# B&R Automation Studio project ULATolo3
Automation Studio 4.7.5.60 SP; technology packages: mapp 5.11.2, mappMotion 5.11.2

## Configuration Config1

CPU X20CP1382, AutomationRuntime B4.73, Build 4.1.2, Safety 0.0, Vc V4.72.0

### Task classes (Cpu.sw)
```
Cyclic#1 (cycle 1200 us, tolerance 0 us):
  Program <- Program.prg
DataObjects: ALHistory
VcDataObjects: Visu <- Visu.dob
Binaries: vccdt, vccbmp, Visu03, vcfile, arial, vccddbox, vcrt, vccstr, vcbclass, vccbtn, vcgclass, vcdsint, vcnet, vccline, vcmgr, vcshared, vcclbox, vccscale, arialbd, vccnum, vcpdvnc, FWRules, vccalarm, vccshape, vcctext, Visu01, vcpdsw, vcfntttf, vccovl, vcalarm, vcpkat, Visu02, udbdef, vccpopup, arsvcreg, vcdsloc, vcchspot, vctcal, TCData, vcpfx20, Config, arconfig, Config_1, asfw, iomap, Role, ashwd, ashwac, sysconf, User, vcpfar00
Libraries: brsystem, sys_lib, runtime, MpAxis, MpCom, MpBase, MpAlarmX, astime, AsBrStr, McBase, McAxis, McAcpAx, asieccon, powerlnk, vcresman, ashw, MpData, DataObj, FileIO
```

### Hardware
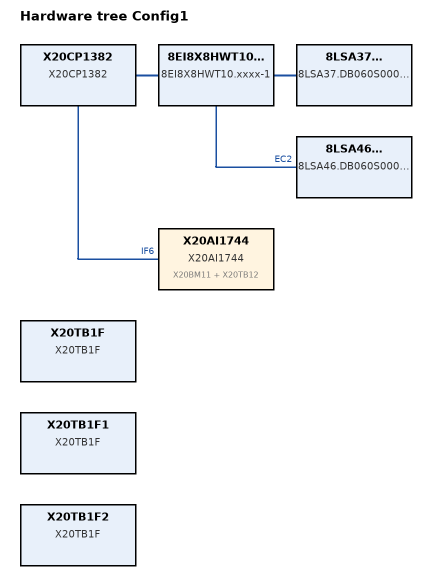
```
8EI8X8HWT10.xxxx-1 : 8EI8X8HWT10.xxxx-1 v2.3.0.3  [PLK2 -> X20CP1382.IF3 [Cable Type=PowerlinkCable, Length=10, Version=1.0.0.2]; EC1 -> 8LSA37.DB060S000-3a.EC; EC2 -> 8LSA46.DB060S000-3.EC; MT2 -> 8LSA46.DB060S000-3.MT]
  MotionTP = Acp10Arnc0
  EnableDNA = on
  EPL_DNA_Head = 0
  EPL_DNA_HubPort = 1
  DriveConfiguration/Module:
    McAcoposTypeID = AcoposP3TConfig
    ActivateACOPOSSimulationOnPLC = 0
  DriveConfiguration/Encoder/EncoderX41:
    InterfaceType = EnDat
  DriveConfiguration/Encoder/EncoderX42:
    InterfaceType = EnDat
  DriveConfiguration/Channel[1]:
    License = 1
  DriveConfiguration/Channel[1]/RealAxis:
    AxisReference = gAxisBasicAxial
  DriveConfiguration/Channel[1]/RealAxis/MechanicalElements/Gearbox:
    InputIsReadOnly = 0
    Input = 40
    OutputIsReadOnly = 0
    Output = 1
  DriveConfiguration/Channel[1]/RealAxis/MechanicalElements/RotaryToLinearTransformation:
    ReferenceDistanceIsReadOnly = 0
    ReferenceDistance = 12.7
  DriveConfiguration/Channel[1]/RealAxis/Controller:
    ModeIsReadOnly = 0
    Mode = PositionController
  DriveConfiguration/Channel[1]/RealAxis/Controller/Mode/Position:
    ProportionalGain = 430
    IntegrationTime = 0.0
    PredictionTime = 0.0004
    TotalDelayTime = 0.0004
  DriveConfiguration/Channel[1]/RealAxis/Controller/Mode/Speed:
    ProportionalGainIsReadOnly = 0
    ProportionalGain = 2.9
    IntegrationTimeIsReadOnly = 0
    IntegrationTime = 0.0
    FilterTimeIsReadOnly = 0
    FilterTime = 0.0
  DriveConfiguration/Channel[1]/RealAxis/Controller/Mode/LoopFilters:
    LoopFilter1 = NotUsed
    LoopFilter2 = NotUsed
    LoopFilter3 = NotUsed
  DriveConfiguration/Channel[1]/RealAxis/Homing:
    Mode = Absolute
  DriveConfiguration/Channel[1]/RealAxis/Homing/Mode:
    Position = 1238.54
  DriveConfiguration/Channel[1]/RealAxis/Homing:
    RestorePositionVariable = 
  DriveConfiguration/Channel[1]/RealAxis/StopReaction:
    Quickstop = DecelerationLimit
    DriveError = DecelerationLimit
  DriveConfiguration/Channel[1]/RealAxis/MovementErrorLimits:
    PositionError = 1.0
    VelocityErrorMonitoring = Automatic1
  DriveConfiguration/Channel[1]/RealAxis:
    JerkFilter = NotUsed
  DriveConfiguration/Channel[1]/RealAxis/DigitalInputs/HomingSwitch:
    Source = NotUsed
    Level = High
  DriveConfiguration/Channel[1]/RealAxis/DigitalInputs/PositiveLimitSwitch:
    Source = NotUsed
    Level = High
  DriveConfiguration/Channel[1]/RealAxis/DigitalInputs/NegativeLimitSwitch:
    Source = NotUsed
    Level = High
  DriveConfiguration/Channel[1]/RealAxis/DigitalInputs/Trigger1:
    Source = X8Trigger1
    Level = High
  DriveConfiguration/Channel[1]/RealAxis/DigitalInputs/Trigger2:
    Source = X8Trigger2
    Level = High
  DriveConfiguration/Channel[1]/RealAxis/DigitalInputs/Quickstop:
    Input = Trigger2
  DriveConfiguration/Channel[1]/RealAxis/Simulation:
    SimulationModeOnPLC = SetValueGeneration
    SimulationModeOnACOPOS = NotUsed
  DriveConfiguration/Channel[2]:
    License = 1
  DriveConfiguration/Channel[2]/RealAxis:
    AxisReference = gAxisBasicSideLoad
  DriveConfiguration/Channel[2]/RealAxis/MechanicalElements/Gearbox:
    InputIsReadOnly = 0
    Input = 1
    OutputIsReadOnly = 0
    Output = 1
  DriveConfiguration/Channel[2]/RealAxis/MechanicalElements/RotaryToLinearTransformation:
    ReferenceDistanceIsReadOnly = 0
    ReferenceDistance = 1
  DriveConfiguration/Channel[2]/RealAxis/Controller:
    ModeIsReadOnly = 0
    Mode = PositionController
  DriveConfiguration/Channel[2]/RealAxis/Controller/Mode/Position:
    ProportionalGain = 50.0
    IntegrationTime = 0.0
    PredictionTime = 0.0004
    TotalDelayTime = 0.0004
  DriveConfiguration/Channel[2]/RealAxis/Controller/Mode/Speed:
    ProportionalGainIsReadOnly = 0
    ProportionalGain = 2.0
    IntegrationTimeIsReadOnly = 0
    IntegrationTime = 0.0
    FilterTimeIsReadOnly = 0
    FilterTime = 0.0
  DriveConfiguration/Channel[2]/RealAxis/Controller/Mode/LoopFilters:
    LoopFilter1 = NotUsed
    LoopFilter2 = NotUsed
    LoopFilter3 = NotUsed
  DriveConfiguration/Channel[2]/RealAxis/Homing:
    Mode = Absolute
  DriveConfiguration/Channel[2]/RealAxis/Homing/Mode:
    Position = 12888.441
  DriveConfiguration/Channel[2]/RealAxis/Homing:
    RestorePositionVariable = 
  DriveConfiguration/Channel[2]/RealAxis/StopReaction:
    Quickstop = DecelerationLimit
    DriveError = DecelerationLimit
  DriveConfiguration/Channel[2]/RealAxis/MovementErrorLimits:
    PositionError = 1.0
    VelocityErrorMonitoring = Automatic1
  DriveConfiguration/Channel[2]/RealAxis:
    JerkFilter = NotUsed
  DriveConfiguration/Channel[2]/RealAxis/DigitalInputs/HomingSwitch:
    Source = NotUsed
    Level = High
  DriveConfiguration/Channel[2]/RealAxis/DigitalInputs/PositiveLimitSwitch:
    Source = NotUsed
    Level = High
  DriveConfiguration/Channel[2]/RealAxis/DigitalInputs/NegativeLimitSwitch:
    Source = NotUsed
    Level = High
  DriveConfiguration/Channel[2]/RealAxis/DigitalInputs/Trigger1:
    Source = X8Trigger1
    Level = High
  DriveConfiguration/Channel[2]/RealAxis/DigitalInputs/Trigger2:
    Source = X8Trigger2
    Level = High
  DriveConfiguration/Channel[2]/RealAxis/DigitalInputs/Quickstop:
    Input = Trigger2
  DriveConfiguration/Channel[2]/RealAxis/Simulation:
    SimulationModeOnPLC = SetValueGeneration
    SimulationModeOnACOPOS = NotUsed
  DriveConfiguration/Channel[3]:
    License = 1
  DriveConfiguration/Channel[3]/RealAxis:
    AxisReference = 
  DriveConfiguration/Channel[3]/RealAxis/MechanicalElements/Gearbox:
    InputIsReadOnly = 0
    Input = 1
    OutputIsReadOnly = 0
    Output = 1
  DriveConfiguration/Channel[3]/RealAxis/MechanicalElements/RotaryToLinearTransformation:
    ReferenceDistanceIsReadOnly = 0
    ReferenceDistance = 1
  DriveConfiguration/Channel[3]/RealAxis/Controller:
    ModeIsReadOnly = 0
    Mode = PositionController
  DriveConfiguration/Channel[3]/RealAxis/Controller/Mode/Position:
    ProportionalGain = 50.0
    IntegrationTime = 0.0
    PredictionTime = 0.0004
    TotalDelayTime = 0.0004
  DriveConfiguration/Channel[3]/RealAxis/Controller/Mode/Speed:
    ProportionalGainIsReadOnly = 0
    ProportionalGain = 2.0
    IntegrationTimeIsReadOnly = 0
    IntegrationTime = 0.0
    FilterTimeIsReadOnly = 0
    FilterTime = 0.0
  DriveConfiguration/Channel[3]/RealAxis/Controller/Mode/LoopFilters:
    LoopFilter1 = NotUsed
    LoopFilter2 = NotUsed
    LoopFilter3 = NotUsed
  DriveConfiguration/Channel[3]/RealAxis/Homing:
    Mode = Direct
  DriveConfiguration/Channel[3]/RealAxis/Homing/Mode:
    Position = 0.0
    ReferencePulse = NotUsed
  DriveConfiguration/Channel[3]/RealAxis/Homing:
    RestorePositionVariable = 
  DriveConfiguration/Channel[3]/RealAxis/StopReaction:
    Quickstop = DecelerationLimit
    DriveError = DecelerationLimit
  DriveConfiguration/Channel[3]/RealAxis/MovementErrorLimits:
    PositionError = 1.0
    VelocityErrorMonitoring = Automatic1
  DriveConfiguration/Channel[3]/RealAxis:
    JerkFilter = NotUsed
  DriveConfiguration/Channel[3]/RealAxis/DigitalInputs/HomingSwitch:
    Source = NotUsed
    Level = High
  DriveConfiguration/Channel[3]/RealAxis/DigitalInputs/PositiveLimitSwitch:
    Source = NotUsed
    Level = High
  DriveConfiguration/Channel[3]/RealAxis/DigitalInputs/NegativeLimitSwitch:
    Source = NotUsed
    Level = High
  DriveConfiguration/Channel[3]/RealAxis/DigitalInputs/Trigger1:
    Source = X8Trigger1
    Level = High
  DriveConfiguration/Channel[3]/RealAxis/DigitalInputs/Trigger2:
    Source = X8Trigger2
    Level = High
  DriveConfiguration/Channel[3]/RealAxis/DigitalInputs/Quickstop:
    Input = Trigger2
  DriveConfiguration/Channel[3]/RealAxis/Simulation:
    SimulationModeOnPLC = SetValueGeneration
    SimulationModeOnACOPOS = NotUsed
8LSA37.DB060S000-3a : 8LSA37.DB060S000-3 v1.0.5.34  [EC -> 8EI8X8HWT10.xxxx-1.EC1; MT -> 8EI8X8HWT10.xxxx-1.MT1]
8LSA46.DB060S000-3 : 8LSA46.DB060S000-3 v2.2.0.0  [EC -> 8EI8X8HWT10.xxxx-1.EC2; MT -> 8EI8X8HWT10.xxxx-1.MT2]
  M1/MotorParameters:
    MOTOR_AMB_TEMP_RATED = 40
  M1/MotorParameters/TemperatureSensor:
    MOTOR_TEMPSENS_LIM = 130
X20AI1744 : X20AI1744 v1.8.4.0  [SS1 -> X20TB12.SS; SL -> X20BM11.SL1]
  Supervision = off
X20BM11 : X20BM11 v1.0.0.1  [X2X1 -> X20CP1382.IF6]
X20CP1382 : X20CP1382 v1.8.0.0  [X1 -> X1.SL; X2 -> X2.SL; X3 -> X3.SL]
  Module X1 (Type=X1, Virtual=true, Version=1.8.0.0)
    Connection (Connector=SS1, TargetModule=X20TB1F, TargetConnector=SS)
    Connection (Connector=SL, TargetModule=X20CP1382, TargetConnector=X1)
  Module X2 (Type=X2, Virtual=true, Version=1.8.0.0)
    Connection (Connector=SS1, TargetModule=X20TB1F1, TargetConnector=SS)
    Connection (Connector=SL, TargetModule=X20CP1382, TargetConnector=X2)
  Module X3 (Type=X3, Virtual=true, Version=1.8.0.0)
    Connection (Connector=SS1, TargetModule=X20TB1F2, TargetConnector=SS)
    Connection (Connector=SL, TargetModule=X20CP1382, TargetConnector=X3)
  Connector IF2:
    ActivateDevice = 1
    Mode = Manual
    InternetAddress = 192.168.1.5
    SubnetMask = 255.255.255.0
    Vnc1
    VncVcObjectName1 = Visu
    VncKeyMappingFile1 = VC\PS2-Keyboard.dis
  Connector IF3:
    CycleTime = 1200
  ConfigurationID = ULATolo3_Config1
  Simulation = 1
  VolatileGlobalPvSize = 6553500
  TimerDeviceType = EPLX2X
  TimerDevice = X20CP1382.IF3
  TaskClassIdleTime = 9600
  Cyclic1Duration = 1200
  Cyclic1Tolerance = 0
  Cyclic1Stack = 65535
  Cyclic2Duration = 20400
  Cyclic2Tolerance = 20400
  Cyclic3Duration = 50400
  Cyclic3Tolerance = 50400
  Cyclic4Duration = 99600
  Cyclic4Tolerance = 99600
  Cyclic5Duration = 200400
  Cyclic5Tolerance = 200400
  Cyclic6Duration = 500400
  Cyclic6Tolerance = 500400
  Cyclic7Duration = 999600
  Cyclic7Tolerance = 999600
  Cyclic8Duration = 9600
  FileDevice1
  FileDeviceName1 = Temp
  FileDevicePath1 = C:\Temp
  FileDevice2
  FileDeviceName2 = PLC
  FileDevicePath2 = F:\
X20TB12 : X20TB12 v1.0.0.0
X20TB1F : X20TB1F v1.0.0.0
X20TB1F1 : X20TB1F v1.0.0.0
X20TB1F2 : X20TB1F v1.0.0.0
```

### IoMap.iom - X20CP1382/IoMap.iom
```iecst
VAR_CONFIG
	::gMain.Input.Physical.StrainGauge AT %ID."X20AI1744".AnalogInput01;
	::gMain.Machine.Motion.PosLimit AT %IX."X1".DigitalInput01;
	::gMain.Machine.Motion.NegLimit AT %IX."X1".DigitalInput02;
END_VAR
```

### Acp10cfg.ncc - X20CP1382/Motion/Acp10cfg.ncc
```
NcConfiguration (Version=5.08.2, NcSwId=Acp10)
  ACP10CF1_typ:
    cnt_nettrc_rec_drive = 1500
    bufsize_trace_upload = 1200
    tc_nc_man_task = Cyclic #1
    glob_pv_as_ncobject = Yes
    ncsys_dl_broadcast = Yes
    ncsys_dl_acp_reset = Yes
    safemc_log_err_to_ax = Yes
    network_init:
      ncsw_init_execute = Yes
      automatic_execute = No
      node_nr_warning = Yes
      net_err_before_ncact = Yes
    nettrc:
      enter_parsecrec = Yes
      enter_ncaction = Yes
      save_ring_startidx = Yes
    cam_prof_download:
      cam_dat_dl_parallel = No
      tc_cam_dl_parallel = Task class for NC Manager task
    plk_if[0]:
      if_name = IF3
      tc_CycDat_PLCopen = Task class for NC Manager task
      mc_broadcast_extdat = No
```

### Acp10map.ncm - X20CP1382/Motion/Acp10map.ncm
```
NcMapping (NcSwId=Acp10, DisabledNodesAreHidden=False)
  NcObject gAxisSideLoad (ModuleId=8EI8X8HWT10.xxxx-1, Type=ncAXIS, Channel=2, AcoposSimulation=Off, InitParameter=gAxis01i, AcoposParameter=gAxis01a, Disabled=FALSE, ModuleDisabled=FALSE)
  NcObject gAxisAxial (ModuleId=8EI8X8HWT10.xxxx-1, Type=ncAXIS, Channel=1, AcoposSimulation=Off, InitParameter=gAxis01i, AcoposParameter=gAxis01a, Disabled=FALSE, ModuleDisabled=FALSE)
  NcObject 8EI4X5HWD10.xxxx-1_ncAXIS3 (ModuleId=8EI8X8HWT10.xxxx-1, Type=ncAXIS, Channel=3, AcoposSimulation=off, Disabled=true, ModuleDisabled=FALSE)
  NcObject 8EI4X5HWD10.xxxx-1_ncV_AXIS2 (ModuleId=8EI8X8HWT10.xxxx-1, Type=ncV_AXIS, Channel=2, Disabled=TRUE, ModuleDisabled=FALSE)
  NcObject 8EI4X5HWD10.xxxx-1_ncV_AXIS1 (ModuleId=8EI8X8HWT10.xxxx-1, Type=ncV_AXIS, Channel=1, Disabled=TRUE, ModuleDisabled=FALSE)
  NcObject 8EI4X5HWD10.xxxx-1_ncV_AXIS3 (ModuleId=8EI8X8HWT10.xxxx-1, Type=ncV_AXIS, Channel=3, AcoposSimulation=off, Disabled=true, ModuleDisabled=FALSE)
```

### Config.mpaxisbasic - X20CP1382/Motion/Config.mpaxisbasic
```
Element gAxisBasicAxial (Type=mpaxisbasic)
  AxisConfiguration = AxisWithConfiguration
    Axis:
      BaseType = 4
      MeasurementUnit = 1
      PeriodSettings:
        Period = 360
      MovementLimits:
        VelocityPositive = 10000.0
        VelocityNegative = 10000.0
        Acceleration = 50000.0
        Deceleration = 50000
        JerkTime = 0.01
        PositionErrorStopLimit = 1000
    Drive:
      Transformation:
        ReferenceDistance = 12.7
      Controller:
        LoopFilters:
          [0]
          [1]
          [2]
  Alarms = MpAlarmX
Element gAxisBasicSideLoad (Type=mpaxisbasic)
  Alarms = MpAlarmX
```

### Axial.axis - X20CP1382/mappMotion/Axial.axis
```
Element gAxisBasicAxial (Type=axis)
  BaseTypeIsReadOnly = 0
  BaseType = LinearBounded
    MeasurementUnit = 5066068
    MeasurementResolutionIsReadOnly = 0
    MeasurementResolution = 0.01
    CountDirectionIsReadOnly = 0
    CountDirection = Standard
  MovementLimitsIsReadOnly = 0
  MovementLimits = Internal
    Position:
      LowerLimitMin = -1.79769313486231E308
      UpperLimitMax = 1.79769313486231E308
      LowerLimit = 388.62
      UpperLimit = 608.6348
    VelocityIsReadOnly = 0
    Velocity:
      VelocityMax = 3.4E38
      Velocity = 50
    AccelerationIsReadOnly = 0
    Acceleration:
      AccelerationMax = 3.4E38
      Acceleration = 75
    DecelerationIsReadOnly = 0
    Deceleration:
      DecelerationMax = 3.4E38
      Deceleration = 75
  Alarms = MpAlarmX
```

### Side.axis - X20CP1382/mappMotion/Side.axis
```
Element gAxisBasicSideLoad (Type=axis)
  BaseTypeIsReadOnly = 0
  BaseType = LinearBounded
    MeasurementUnit = 5066068
    MeasurementResolutionIsReadOnly = 0
    MeasurementResolution = 0.01
    CountDirectionIsReadOnly = 0
    CountDirection = Standard
  MovementLimitsIsReadOnly = 0
  MovementLimits = Internal
    Position:
      LowerLimitMin = -1.79769313486231E308
      UpperLimitMax = 1.79769313486231E308
      LowerLimit = -1000.0
      UpperLimit = 1000.0
    VelocityIsReadOnly = 0
    Velocity:
      VelocityMax = 3.4E38
      Velocity = 25
    AccelerationIsReadOnly = 0
    Acceleration:
      AccelerationMax = 3.4E38
      Acceleration = 75
    DecelerationIsReadOnly = 0
    Deceleration:
      DecelerationMax = 3.4E38
      Deceleration = 75
  Alarms = MpAlarmX
```

### Config.mpdatarecorder - X20CP1382/mappServices/Config.mpdatarecorder
```
Element gDataRecorder (Type=mpdatarecorder)
  Alarms = MpAlarmX
```

### Config_1.mpalarmxcore - X20CP1382/mappServices/Config_1.mpalarmxcore
```
Element gAlarmXCore (Type=mpalarmxcore)
```

## Logical view

Binary libraries used (declarations not repeated): operator, runtime, astime, AsIecCon, brsystem, sys_lib, AsBrStr, McBase 5.11.2, McAxis 5.11.2, MpBase 5.11.0, MpAlarmX 5.11.2, MpCom 5.11.2, MpAxis 5.11.2, McAcpAx 5.11.2, MpData 5.11.2, DataObj, FileIO, Acp10_MC 5.10.1, Acp10man 5.10.1, Acp10par 5.10.1, NcGlobal 5.10.1

### Global.typ - Global data types
```iecst
TYPE
	Alarm_Type : 	STRUCT
		MpAlarmXListUI_FB : MpAlarmXListUI;
		MpAlarmXAcknowledgeAll_FB : MpAlarmXAcknowledgeAll;
		MpAlarmXListUISetupType : MpAlarmXListUISetupType;
		MpAlarmXListUIConnectType : MpAlarmXListUIConnectType;
		AlarmPopupControl : USINT;
		MpAlarmXCore_FB : MpAlarmXCore;
	END_STRUCT;
	InputPhysical_Type : 	STRUCT
		LoadtoTorqueScaleFactor : REAL;
		StrainGauge : DINT;
	END_STRUCT;
	Output_Type : 	STRUCT
		Physical : OutputPhysical_Type;
		Vis : OutputVis_Type;
	END_STRUCT;
	OutputVis_Type : 	STRUCT
		DisplayedForceFeedback : REAL;
		StatusLED : USINT;
		LoadCellScaleFactor : REAL;
		CalculatedForce : REAL;
	END_STRUCT;
	OutputPhysical_Type : 	STRUCT
		New_Member : USINT;
	END_STRUCT;
	InputVis_Type : 	STRUCT
		NumberofCycles : USINT;
		ManualCommandedAxialPosition : REAL;
		ManualReturnButton : BOOL;
		ManualCommandedSideLoad : REAL;
		AxisSelector : USINT;
		JogNeg : BOOL;
		JogPos : BOOL;
		ManualMoveButton : BOOL;
		StartProgramButton : BOOL;
		NominalPosition : REAL;
		AutoCommandedAxialPosition : REAL;
		PowerOnButtonVisibility : USINT;
		JogButtonVisibility : USINT;
		StopButtonVisibility : USINT;
		StartButtonVisability : USINT;
		EStopPopup : USINT;
		EStop : BOOL;
		PowerOnAll : BOOL;
		OscillationDistance : REAL;
		ManualStopButtonVis : UINT;
		ConfirmPopup : USINT;
		ManualGoButtonVis : UINT;
	END_STRUCT;
	Input_Type : 	STRUCT
		Physical : InputPhysical_Type;
		Vis : InputVis_Type;
	END_STRUCT;
	Motion_Type : 	STRUCT
		MpAxisBasicPar : ARRAY[Axial..SideLoad]OF MpAxisBasicParType;
		Mc_StopFB : ARRAY[Axial..SideLoad]OF MC_Stop;
		MpAxisBasic_FB : ARRAY[Axial..SideLoad]OF MpAxisBasic;
		Error : BOOL;
		HomeAll : BOOL;
		IsHomedAll : BOOL;
		AllAxisReady : BOOL;
		ErrorResetAll : BOOL;
		SideLoad : SideLoad_Type;
		AxialMove : AxialMove_Type;
		IsPoweredAll : BOOL;
		AtNominalFlag : BOOL;
	END_STRUCT;
	Machine_Type : 	STRUCT
		State : StateEnum;
		Alarm : Alarm_Type;
		Motion : Motion_Type;
	END_STRUCT;
	Main_Type : 	STRUCT
		Output : Output_Type;
		Input : Input_Type;
		Machine : Machine_Type;
		Services : Services_Type;
	END_STRUCT;
	SideLoad_Type : 	STRUCT
		ScalingFactor : REAL;
		EnableCyclicTorque : BOOL;
		TorqueScaled : REAL;
		MC_TorqueControl_FB : MC_TorqueControl;
		MC_MoveAdditive_SideLoad : MC_MoveAdditive;
	END_STRUCT;
	AxialMove_Type : 	STRUCT
		Amax : REAL;
		TotalDistance : REAL;
		Vmax : REAL;
		TotalTime : REAL;
		CyclicCommandedPosition : REAL;
		CycleAmplitude : REAL;
		FirstMovementFlag : BOOL;
		ChangeDirectionFlag : BOOL;
		CycleCount : UDINT;
		PositionOffset : REAL;
		MC_MoveAdditive_Axial : MC_MoveAdditive;
	END_STRUCT;
	AxisEnum :
		(
		SideLoad := 1,
		Axial := 0
		);
	StateEnum :
		(
		Running := 6,
		Idle := 5,
		WaitingForPowerOn := 4,
		Homing := 3,
		AxisReady := 2,
		Init := 1,
		Error := 0
		);
	Services_Type : 	STRUCT
		MpDataRegPar : MpDataRegPar;
		MpDataRecorder_FB : MpDataRecorder;
	END_STRUCT;
END_TYPE
```

### Global.var - Global variables
```iecst
VAR
	gMain : Main_Type;
	i0 : USINT;
END_VAR
```

### Package Logical/Libraries - Global libraries

- Visualisation Logical/Visu (not shown)

### Program Logical/Program (IEC)

#### Variables.var
```iecst
VAR CONSTANT
	MAX_TORQUE : REAL := 169.477;
END_VAR
```

#### Main.st
```iecst
PROGRAM _INIT

//
//		gMain.Machine.Motion.AxialMove.CycleAmplitude:=12.7;
//		gMain.Machine.Motion.AxialMove.TotalTime:=0.0825;
//		gMain.Machine.Motion.AxialMove.TotalDistance:=gMain.Machine.Motion.AxialMove.CycleAmplitude*2;
//		gMain.Machine.Motion.AxialMove.PositionOffset:=18.2*25.4;
//
//	gMain.Machine.Motion.Mc_StopFB[Axial](Axis := ADR(gAxisAxial), Deceleration := 50000);
//	gMain.Machine.Motion.Mc_StopFB[SideLoad](Axis := ADR(gAxisSideLoad), Deceleration := 50000);
//
//		// Velocity AND Acceleration Calculations FOR Axial MOVE
//		IF gMain.Machine.Motion.AxialMove.TotalTime<>0.0 THEN
//			gMain.Machine.Motion.AxialMove.Vmax:=ABS(gMain.Machine.Motion.AxialMove.TotalDistance/(0.5*(gMain.Machine.Motion.AxialMove.TotalTime)));
//			gMain.Machine.Motion.AxialMove.Amax:=ABS(gMain.Machine.Motion.AxialMove.Vmax/(0.5*gMain.Machine.Motion.AxialMove.TotalTime));
//		END_IF;
//
//	gMain.Machine.Motion.MpAxisBasicPar[Axial].Acceleration:=gMain.Machine.Motion.AxialMove.Amax;
//	gMain.Machine.Motion.MpAxisBasicPar[Axial].Deceleration:=gMain.Machine.Motion.AxialMove.Amax;
//	gMain.Machine.Motion.MpAxisBasicPar[Axial].Velocity:=gMain.Machine.Motion.AxialMove.Vmax;
//
//
//
//	gMain.Machine.Motion.MpAxisBasicPar[Axial].Home.Mode:=mpAXIS_HOME_MODE_ABSOLUTE;
//	gMain.Machine.Motion.MpAxisBasicPar[Axial].Home.Position:=1238.54;						//0 position is -610.77
//
//	gMain.Machine.Motion.MpAxisBasicPar[SideLoad].Home.Mode:=mpAXIS_HOME_MODE_ABSOLUTE;
//	gMain.Machine.Motion.MpAxisBasicPar[SideLoad].Home.Position:=12888.441;

	gMain.Machine.Motion.MpAxisBasic_FB[Axial].MpLink := ADR(gAxisBasicAxial);
	gMain.Machine.Motion.MpAxisBasic_FB[Axial].Enable := TRUE;
	gMain.Machine.Motion.MpAxisBasic_FB[Axial].Parameters := ADR(gMain.Machine.Motion.MpAxisBasicPar[Axial]);
	//gMain.Machine.Motion.MpAxisBasic_FB[Axial].Axis := ADR(gAxisAxial);

	gMain.Machine.Motion.MpAxisBasic_FB[SideLoad].MpLink :=ADR(gAxisBasicSideLoad);
	gMain.Machine.Motion.MpAxisBasic_FB[SideLoad].Enable := TRUE;
	gMain.Machine.Motion.MpAxisBasic_FB[SideLoad].Parameters := ADR(gMain.Machine.Motion.MpAxisBasicPar[SideLoad]);
	//gMain.Machine.Motion.MpAxisBasic_FB[SideLoad].Axis := ADR(gAxisSideLoad);

	gMain.Machine.Motion.SideLoad.MC_TorqueControl_FB.Axis := ADR(gAxisBasicSideLoad);
	gMain.Machine.Motion.SideLoad.MC_TorqueControl_FB.TorqueRamp := 0.3;
	gMain.Machine.Motion.SideLoad.MC_TorqueControl_FB.Velocity := 10;
	gMain.Machine.Motion.SideLoad.MC_TorqueControl_FB.Acceleration := 10;

	gMain.Machine.Alarm.MpAlarmXCore_FB(MpLink :=ADR(gAlarmXCore),Enable := TRUE);
	gMain.Machine.Alarm.MpAlarmXListUI_FB(MpLink := ADR(gAlarmXCore), Enable := TRUE, UISetup := gMain.Machine.Alarm.MpAlarmXListUISetupType, UIConnect := ADR(gMain.Machine.Alarm.MpAlarmXListUIConnectType));

//	gMain.Machine.Motion.MpAxisBasicPar[SideLoad].CyclicRead.TorqueMode:=mpAXIS_READ_CYCLIC;

	gMain.Output.Vis.LoadCellScaleFactor:= (100.0/-307482);
	gMain.Machine.Motion.SideLoad.ScalingFactor := 0.0034;

	gMain.Machine.Motion.MpAxisBasicPar[Axial].Jog.Velocity:=25.4;

	//Data Logging
	gMain.Services.MpDataRecorder_FB.DeviceName := ADR('Temp');
	gMain.Services.MpDataRecorder_FB.RecordMode := mpDATA_RECORD_MODE_VALUE;
	gMain.Services.MpDataRecorder_FB.MpLink := ADR(gDataRecorder);
	gMain.Services.MpDataRecorder_FB.Enable :=  TRUE;

	gMain.Services.MpDataRegPar.MpLink := ADR(gDataRecorder);
	gMain.Services.MpDataRegPar.Enable := TRUE;
	gMain.Services.MpDataRegPar.PVName := ADR('gMain.Input.Vis.StartProgramButton');

	//Popup Vis
	gMain.Input.Vis.ConfirmPopup := TRUE;
END_PROGRAM

PROGRAM _CYCLIC
	gMain.Machine.Motion.AllAxisReady :=TRUE;
	gMain.Machine.Motion.IsHomedAll := TRUE;
	gMain.Machine.Motion.IsPoweredAll := TRUE;
	gMain.Machine.Motion.Error := FALSE;
	//gMain.Machine.Motion.AxialMove.MC_MoveAdditive_Axial.Execute:=FALSE;

	//Check State Loop
	FOR i0:=DINT_TO_USINT(Axial) TO DINT_TO_USINT(SideLoad) DO
		IF NOT gMain.Machine.Motion.MpAxisBasic_FB[i0].Info.ReadyToPowerOn AND NOT gMain.Machine.Motion.MpAxisBasic_FB[i0].Info.ReadyToPowerOn THEN //If not axis initilaized and not ready to power on
			gMain.Machine.Motion.AllAxisReady := FALSE;  																						   //Then set DrivesReady to FALSE
		END_IF;
		IF gMain.Machine.Motion.MpAxisBasic_FB[i0].IsHomed = FALSE THEN																				//If single axis is not homed
			gMain.Machine.Motion.IsHomedAll := FALSE;																								//Then IsHomedAll is FALSE
		END_IF;
		IF gMain.Machine.Motion.MpAxisBasic_FB[i0].PowerOn = FALSE THEN																				//If drive PowerOn is FALSE for single axis
			gMain.Machine.Motion.IsPoweredAll := FALSE;																								//Then IsPoweredAll is FALSE
		END_IF;
		IF gMain.Machine.Motion.MpAxisBasic_FB[i0].Error THEN
			gMain.Machine.Motion.Error:=TRUE;
		END_IF;
	END_FOR;

	//Machine State Case Statement
	CASE gMain.Machine.State OF
		Error:
			IF gMain.Machine.Motion.Error THEN
			ELSE
				gMain.Machine.State:=Init;
			END_IF;
			gMain.Input.Vis.PowerOnAll:=FALSE;
			gMain.Output.Vis.StatusLED:=0;
			gMain.Services.MpDataRecorder_FB.Record := FALSE;
		Init:
			IF gMain.Machine.Motion.Error THEN
				gMain.Machine.State:=Error;
			ELSIF gMain.Machine.Motion.AllAxisReady THEN
				gMain.Machine.Motion.HomeAll:=TRUE;
				gMain.Machine.State:=Homing;
			END_IF;
		Homing:
			IF gMain.Machine.Motion.Error THEN
				gMain.Machine.State:=Error;
			ELSIF gMain.Machine.Motion.IsHomedAll THEN
				gMain.Machine.Motion.HomeAll:=FALSE;
				gMain.Machine.State:=WaitingForPowerOn;
			END_IF;
		WaitingForPowerOn:
			IF gMain.Machine.Motion.Error THEN
				gMain.Machine.State:=Error;
			ELSIF NOT gMain.Machine.Motion.IsHomedAll THEN
				gMain.Machine.State:=Init;
			ELSIF gMain.Machine.Motion.IsPoweredAll THEN
				gMain.Machine.State:=Idle;
			END_IF;
			gMain.Output.Vis.StatusLED:=1;
			//			gMain.Input.Vis.PowerButtonVisibility:=FALSE;
			//			gMain.Input.Vis.StopProgramButton:=FALSE;
			//			gMain.Input.Vis.StartProgramButton:=FALSE;
			//			gMain.Input.Vis.PauseProgramButton :=FALSE;
			//			gMain.Machine.Motion.ProgramRunningFlag:=FALSE;
			//			gMain.Machine.Motion.McMoveAbsoluteFB.Execute:=FALSE;
			//			gMain.Output.Vis.CycleCount:=Error;
		Idle:
			IF gMain.Machine.Motion.Error THEN
				gMain.Machine.State:=Error;
			ELSIF gMain.Machine.Motion.IsPoweredAll=FALSE THEN
				gMain.Machine.State:=WaitingForPowerOn;
			ELSIF gMain.Input.Vis.StartProgramButton THEN
				gMain.Machine.State:=Running;
			END_IF;
			gMain.Output.Vis.StatusLED:=2;
			gMain.Services.MpDataRecorder_FB.Record := TRUE;
			//Jog Logic
			IF gMain.Input.Vis.AxisSelector = 0 THEN
				gMain.Machine.Motion.MpAxisBasic_FB[0].JogPositive:=gMain.Input.Vis.JogNeg;
				gMain.Machine.Motion.MpAxisBasic_FB[0].JogNegative:=gMain.Input.Vis.JogPos;
			ELSE
				gMain.Machine.Motion.MpAxisBasic_FB[1].JogPositive:=gMain.Input.Vis.JogPos;
				gMain.Machine.Motion.MpAxisBasic_FB[1].JogNegative:=gMain.Input.Vis.JogNeg;
			END_IF;

			//Manual Move Logic

			gMain.Machine.Motion.AxialMove.MC_MoveAdditive_Axial.Execute:=gMain.Input.Vis.ManualMoveButton;
			gMain.Machine.Motion.AxialMove.MC_MoveAdditive_Axial.Distance:=-gMain.Input.Vis.ManualCommandedAxialPosition;

			gMain.Machine.Motion.SideLoad.TorqueScaled := gMain.Input.Vis.ManualCommandedSideLoad*gMain.Machine.Motion.SideLoad.ScalingFactor;
			gMain.Machine.Motion.SideLoad.EnableCyclicTorque := gMain.Input.Vis.ManualMoveButton;

		Running:
			IF gMain.Machine.Motion.Error THEN
				gMain.Machine.State:=Error;
			ELSIF gMain.Machine.Motion.IsPoweredAll=FALSE THEN
				gMain.Machine.State:=WaitingForPowerOn;
			ELSIF NOT gMain.Input.Vis.StartProgramButton THEN
				gMain.Machine.State:=Idle;
			END_IF;

	END_CASE;

	//Alarms
	gMain.Machine.Alarm.MpAlarmXCore_FB(ErrorReset := gMain.Machine.Motion.ErrorResetAll);
	gMain.Machine.Alarm.MpAlarmXListUI_FB(ErrorReset := gMain.Machine.Motion.ErrorResetAll);
	gMain.Machine.Alarm.AlarmPopupControl:=BOOL_TO_USINT(NOT UDINT_TO_BOOL(gMain.Machine.Alarm.MpAlarmXCore_FB.PendingAlarms));

	//Button Visibility
	gMain.Input.Vis.PowerOnButtonVisibility:=NOT (gMain.Machine.Motion.AllAxisReady);
	gMain.Input.Vis.StartButtonVisability:= NOT (gMain.Machine.Motion.IsPoweredAll AND NOT gMain.Input.Vis.StartProgramButton);
	gMain.Input.Vis.StopButtonVisibility:= NOT gMain.Input.Vis.StartProgramButton;
	gMain.Input.Vis.ManualGoButtonVis := gMain.Input.Vis.ManualMoveButton;
	gMain.Input.Vis.ManualStopButtonVis := NOT  gMain.Input.Vis.ManualMoveButton;

	//Axial Movement
	IF gMain.Machine.Motion.SideLoad.MC_TorqueControl_FB.InTorque THEN
		gMain.Machine.Motion.MpAxisBasic_FB[SideLoad].MoveAbsolute := FALSE;

		IF NOT gMain.Machine.Motion.AxialMove.ChangeDirectionFlag AND gMain.Input.Vis.StartProgramButton AND gMain.Machine.Motion.AxialMove.CycleCount<gMain.Input.Vis.NumberofCycles AND gMain.Machine.Motion.AxialMove.FirstMovementFlag THEN
			IF gMain.Machine.Motion.AxialMove.MC_MoveAdditive_Axial.Done THEN
				gMain.Machine.Motion.AxialMove.ChangeDirectionFlag:=1;
				gMain.Machine.Motion.AxialMove.MC_MoveAdditive_Axial.Execute:=FALSE;
			ELSE
				gMain.Machine.Motion.AxialMove.MC_MoveAdditive_Axial.Execute:=TRUE;
				gMain.Machine.Motion.AxialMove.MC_MoveAdditive_Axial.Distance:=gMain.Input.Vis.OscillationDistance*2;
			END_IF;
		ELSIF gMain.Machine.Motion.AxialMove.ChangeDirectionFlag AND gMain.Input.Vis.StartProgramButton AND gMain.Machine.Motion.AxialMove.CycleCount<gMain.Input.Vis.NumberofCycles (*AND gMain.Machine.Motion.SideLoad.MpAxisCyclicSet_FB.Info.TorqueControl.InTorque*) THEN
			IF gMain.Machine.Motion.AxialMove.MC_MoveAdditive_Axial.Done THEN
				gMain.Machine.Motion.AxialMove.ChangeDirectionFlag:=0;
				gMain.Machine.Motion.AxialMove.MC_MoveAdditive_Axial.Execute:=FALSE;
				gMain.Machine.Motion.AxialMove.CycleCount:=gMain.Machine.Motion.AxialMove.CycleCount+1;
			ELSE
				gMain.Machine.Motion.AxialMove.MC_MoveAdditive_Axial.Execute:=TRUE;
				gMain.Machine.Motion.AxialMove.MC_MoveAdditive_Axial.Distance:=-gMain.Input.Vis.OscillationDistance*2;
			END_IF;
		ELSIF NOT gMain.Machine.Motion.AxialMove.ChangeDirectionFlag AND gMain.Input.Vis.StartProgramButton AND gMain.Machine.Motion.AxialMove.CycleCount<gMain.Input.Vis.NumberofCycles AND NOT gMain.Machine.Motion.AxialMove.FirstMovementFlag THEN
			IF gMain.Machine.Motion.AxialMove.MC_MoveAdditive_Axial.Done THEN
				gMain.Machine.Motion.AxialMove.ChangeDirectionFlag:=1;
				gMain.Machine.Motion.AxialMove.FirstMovementFlag:=1;
				gMain.Machine.Motion.AxialMove.MC_MoveAdditive_Axial.Execute:=FALSE;
			ELSE
				gMain.Machine.Motion.AxialMove.MC_MoveAdditive_Axial.Execute:=TRUE;
				gMain.Machine.Motion.AxialMove.MC_MoveAdditive_Axial.Distance:=gMain.Input.Vis.OscillationDistance;
			END_IF;

		ELSIF gMain.Machine.Motion.AxialMove.CycleCount=gMain.Input.Vis.NumberofCycles AND gMain.Input.Vis.StartProgramButton THEN
			IF gMain.Machine.Motion.AxialMove.MC_MoveAdditive_Axial.Done THEN
				gMain.Machine.Motion.AxialMove.MC_MoveAdditive_Axial.Execute:=FALSE;

				gMain.Input.Vis.StartProgramButton:=0;
				gMain.Machine.Motion.AxialMove.CycleCount:=0;
				gMain.Machine.Motion.AxialMove.ChangeDirectionFlag:=0;
				gMain.Machine.Motion.AxialMove.FirstMovementFlag:=0;
				gMain.Machine.Motion.MpAxisBasic_FB[SideLoad].MoveAbsolute := TRUE;
			ELSE
				gMain.Machine.Motion.AxialMove.MC_MoveAdditive_Axial.Execute:=TRUE;
				gMain.Machine.Motion.AxialMove.MC_MoveAdditive_Axial.Distance:=gMain.Input.Vis.OscillationDistance;
			END_IF;
		END_IF;
	END_IF;

	//Torque Control Side Load
	gMain.Input.Vis.NominalPosition :=LREAL_TO_REAL(gMain.Machine.Motion.MpAxisBasic_FB[Axial].Position)+gMain.Input.Vis.AutoCommandedAxialPosition;
	gMain.Output.Vis.DisplayedForceFeedback:= (gMain.Input.Physical.StrainGauge-16275)*gMain.Output.Vis.LoadCellScaleFactor;
	//gMain.Machine.Motion.SideLoad.TorqueScaled:=gMain.Output.Vis.DisplayedForceFeedback*gMain.Machine.Motion.SideLoad.ScalingFactor;

	IF gMain.Input.Vis.StartProgramButton AND NOT gMain.Machine.Motion.AtNominalFlag THEN
		//Force Calculation
		gMain.Output.Vis.CalculatedForce:=-1957.5693+(240.0518*(gMain.Input.Vis.NominalPosition/25.4))-(6.3530*((gMain.Input.Vis.NominalPosition/25.4))**2);
		gMain.Machine.Motion.SideLoad.TorqueScaled:=gMain.Output.Vis.CalculatedForce*gMain.Machine.Motion.SideLoad.ScalingFactor;

		gMain.Machine.Motion.AxialMove.MC_MoveAdditive_Axial.Distance := gMain.Input.Vis.AutoCommandedAxialPosition;
		gMain.Machine.Motion.AxialMove.MC_MoveAdditive_Axial.Execute := TRUE;
		IF gMain.Machine.Motion.AxialMove.MC_MoveAdditive_Axial.Done THEN
			gMain.Machine.Motion.AtNominalFlag := TRUE;
			gMain.Machine.Motion.AxialMove.MC_MoveAdditive_Axial.Execute := FALSE;
		END_IF;
	ELSIF gMain.Input.Vis.StartProgramButton AND gMain.Machine.Motion.AtNominalFlag THEN
		gMain.Input.Vis.ConfirmPopup := TRUE;
		gMain.Machine.Motion.SideLoad.EnableCyclicTorque:=TRUE;
	ELSIF NOT gMain.Input.Vis.StartProgramButton AND NOT gMain.Input.Vis.ManualMoveButton THEN
		gMain.Machine.Motion.SideLoad.EnableCyclicTorque:=FALSE;
		gMain.Machine.Motion.AtNominalFlag := FALSE;
		gMain.Machine.Motion.AxialMove.MC_MoveAdditive_Axial.Execute := FALSE;
	END_IF;

	//EStop Logic
	IF gMain.Input.Vis.EStop THEN
		gMain.Input.Vis.EStopPopup:=0;
		FOR i0:=DINT_TO_USINT(Axial) TO DINT_TO_USINT(SideLoad) DO

			gMain.Input.Vis.PowerOnAll:=FALSE;
			gMain.Machine.Motion.SideLoad.EnableCyclicTorque:=FALSE;
			gMain.Machine.Motion.AxialMove.MC_MoveAdditive_Axial.Execute:=FALSE;
			gMain.Input.Vis.StartProgramButton:=0;
			gMain.Machine.Motion.AxialMove.CycleCount:=0;
			gMain.Machine.Motion.AxialMove.FirstMovementFlag:=0;
		END_FOR;

	ELSE
		gMain.Input.Vis.EStopPopup:=1;
		gMain.Machine.Motion.Mc_StopFB[i0].Execute:=FALSE;
	END_IF;

	//Data Logging
	IF gMain.Services.MpDataRecorder_FB.Error THEN
		gMain.Services.MpDataRecorder_FB.ErrorReset := TRUE;
		gMain.Services.MpDataRecorder_FB.Record := FALSE;
	ELSIF gMain.Services.MpDataRecorder_FB.ErrorReset OR (gMain.Machine.State > Homing AND NOT gMain.Services.MpDataRecorder_FB.Record) THEN
		gMain.Services.MpDataRecorder_FB.ErrorReset := FALSE;
		gMain.Services.MpDataRecorder_FB.Record := TRUE;
	END_IF;

	gMain.Services.MpDataRegPar();
	gMain.Services.MpDataRecorder_FB();

	//Axial Move Absolute
	IF gMain.Machine.Motion.SideLoad.TorqueScaled > MAX_TORQUE THEN
		gMain.Machine.Motion.SideLoad.TorqueScaled := MAX_TORQUE;
	END_IF;

	gMain.Machine.Motion.SideLoad.MC_TorqueControl_FB(Execute := gMain.Machine.Motion.SideLoad.EnableCyclicTorque, Torque := gMain.Machine.Motion.SideLoad.TorqueScaled);

	//Move Addative
	gMain.Machine.Motion.AxialMove.MC_MoveAdditive_Axial(Velocity := 25.4, Acceleration := 25.4, Deceleration := 25.4);
	gMain.Machine.Motion.SideLoad.MC_MoveAdditive_SideLoad(Velocity := 12.7, Acceleration := 25.4, Deceleration := 25.4);

	//Motion Function Call
	FOR i0:=DINT_TO_USINT(Axial) TO DINT_TO_USINT(SideLoad) DO
		gMain.Machine.Motion.MpAxisBasic_FB[i0](ErrorReset := gMain.Machine.Motion.ErrorResetAll, Power := gMain.Input.Vis.PowerOnAll, Home := gMain.Machine.Motion.HomeAll);
		gMain.Machine.Motion.Mc_StopFB[i0]();
	END_FOR;

END_PROGRAM
PROGRAM _EXIT
	gMain.Machine.Motion.MpAxisBasic_FB[Axial](Enable := FALSE);
	gMain.Machine.Motion.MpAxisBasic_FB[SideLoad](Enable := FALSE);

END_PROGRAM
```
